// TIA Portal V17 export
// export: Created 2022-07-05T08:45:17.2421703Z, ExportSetting WithDefaults, DisplayName Totally Integrated Automation Portal, DisplayVersion V17, DisplayName TIA Portal Openness, DisplayVersion V17, DisplayName TIA Portal Version Control Interface, DisplayVersion V17, DisplayName STEP 7 Professional, DisplayVersion V17, DisplayName STEP 7 Safety, DisplayVersion V17, DisplayName WinCC Advanced, DisplayVersion V17
TYPE "namespaceType"
// stored: IsFailsafeCompliant false
   STRUCT
      NamespaceURIs { ExternalAccessible := 'False'; ExternalVisible := 'False'; ExternalWritable := 'False'} : Array[0..0] of WString;
      ServerNamespaceIndexes { ExternalAccessible := 'False'; ExternalVisible := 'False'; ExternalWritable := 'False'} : Array[0..0] of UInt;
      NamespaceStatusList { ExternalAccessible := 'False'; ExternalVisible := 'False'; ExternalWritable := 'False'} : Array[0..0] of DWord;
      NamespaceCount { ExternalAccessible := 'False'; ExternalVisible := 'False'; ExternalWritable := 'False'} : UInt;
   END_STRUCT;
   // NamespaceURIs[0] := WSTRING#'http://www.siemens.com/simatic-s7-opcua';
END_TYPE
